PROGRAM MAIN
VAR
	CurrentNum AT%IB10:INT;
	CurrentVoltage : REAL;
	
	Overname : BOOL;
	Autonoom : BOOL;
	AutonomousButton : BOOL;
END_VAR

IF Autonoom THEN
	CurrentVoltage := CurrentNum/6552;
	Autonoom R= CurrentVoltage > 1;
END_IF
Autonoom S= AutonomousButton;

END_PROGRAM

(* stored: Version 1.1.0.1, ProductVersion 3.1.4024.3
   POU MAIN: Id {2db006ed-2e8f-4f8a-ade4-51905413193e}, SpecialFunc None *)
